SUBAPPLICATION Uebung_103 (* DigitalInput_I1 auf DigitalOutput_Q1, mit Plug and Socket und DEMUX *)
  (* Standard: 61499-2; Description: Copyright (c) 2023 Meisterschulen am Ostbahnhof This program and the accompanying materials are made available under the terms of the Eclipse Public License 2.0 which is available at https://www.eclipse.org/legal/epl-2.0/ SPDX-License-Identifier: EPL-2.0 *)
  (* Version 1.0, 2023-10-23, Franz Höpfinger, Meisterschulen am Ostbahnhof *)
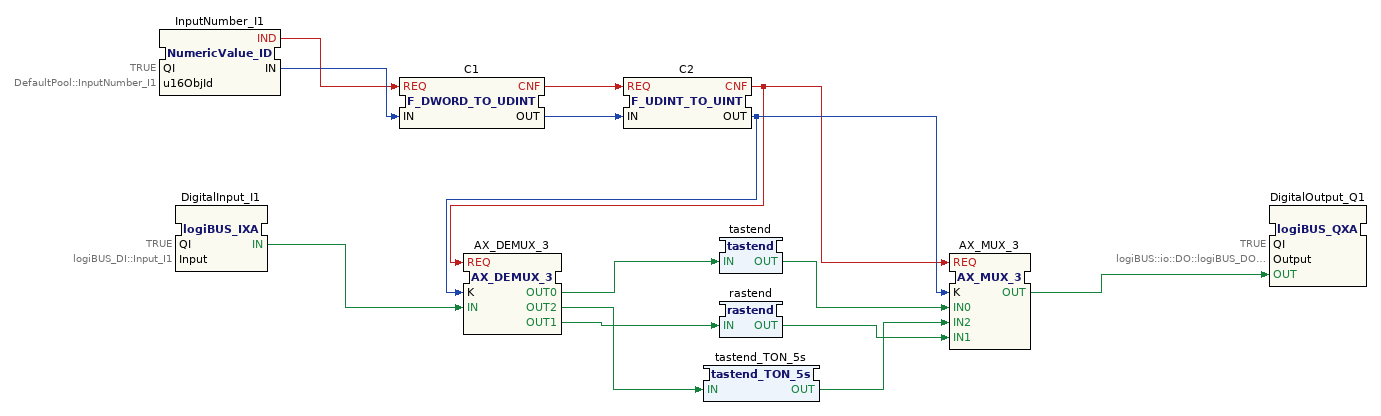
  FBS
    DigitalInput_I1 : logiBUS_IXA(QI := TRUE, Input := logiBUS_DI::Input_I1);
    DigitalOutput_Q1 : logiBUS_QXA(QI := TRUE, Output := logiBUS::io::DO::logiBUS_DO::Output_Q1);
    AX_DEMUX_3 : AX_DEMUX_3;
    AX_MUX_3 : AX_MUX_3;
    InputNumber_I1 : NumericValue_ID(QI := TRUE, u16ObjId := DefaultPool::InputNumber_I1);
    C1 : iec61131::conversion::F_DWORD_TO_UDINT;
    C2 : iec61131::conversion::F_UDINT_TO_UINT;
  END_FBS
  SUBAPPS
    rastend : FBs::Uebungen::Uebung_103::subapp::rastend;
    tastend : FBs::Uebungen::Uebung_103::subapp::tastend;
    tastend_TON_5s : FBs::Uebungen::Uebung_103::subapp::tastend_TON_5s;
  END_SUBAPPS
  EVENT_CONNECTIONS
    InputNumber_I1.IND TO C1.REQ;
    C1.CNF TO C2.REQ;
    C2.CNF TO AX_DEMUX_3.REQ;
    C2.CNF TO AX_MUX_3.REQ;
  END_CONNECTIONS
  DATA_CONNECTIONS
    InputNumber_I1.IN TO C1.IN;
    C1.OUT TO C2.IN;
    C2.OUT TO AX_DEMUX_3.K;
    C2.OUT TO AX_MUX_3.K;
  END_CONNECTIONS
  ADAPTER_CONNECTIONS
    AX_MUX_3.OUT TO DigitalOutput_Q1.OUT;
    DigitalInput_I1.IN TO AX_DEMUX_3.IN;
    AX_DEMUX_3.OUT0 TO tastend.IN;
    tastend.OUT TO AX_MUX_3.IN0;
    AX_DEMUX_3.OUT2 TO tastend_TON_5s.IN;
    tastend_TON_5s.OUT TO AX_MUX_3.IN2;
    rastend.OUT TO AX_MUX_3.IN1;
    AX_DEMUX_3.OUT1 TO rastend.IN;
  END_CONNECTIONS
END_SUBAPPLICATION
